% RSLogix 500 project SARANARA_BAK012.RSS, saved by version 8.10.00.18 %
PROJECT "SARANARA"    % processor: MicroLogix 1200 %

PROGRAM FILES
  LAD 2   7 rungs

DATA FILES
  O0 OUTPUT  4 elements
  I1 INPUT  4 elements
  S2 STATUS  66 elements
  B3 BINARY  1 elements
  T4 TIMER  1 elements
  C5 COUNTER  2 elements
  R6 CONTROL  1 elements
  N7 INTEGER  1 elements

LADDER 2
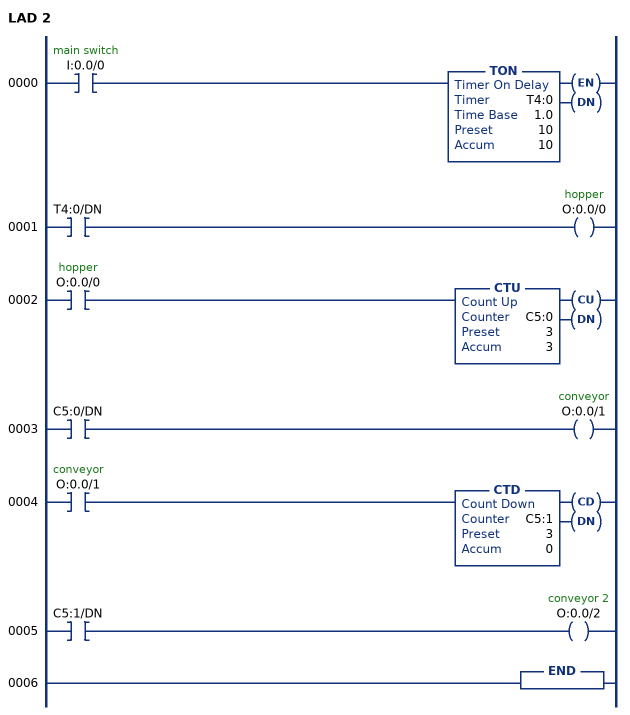
% Rung: 0 %
SOR XIC I:0.0/0 TON T4:0 1.0 10 10 EOR
%   I:0.0/0  "main switch" %
% Rung: 1 %
SOR XIC T4:0/DN OTE O:0.0/0 EOR
%   O:0.0/0  "hopper" %
% Rung: 2 %
SOR XIC O:0.0/0 CTU C5:0 3 3 EOR
%   O:0.0/0  "hopper" %
% Rung: 3 %
SOR XIC C5:0/DN OTE O:0.0/1 EOR
%   O:0.0/1  "conveyor" %
% Rung: 4 %
SOR XIC O:0.0/1 CTD C5:1 3 0 EOR
%   O:0.0/1  "conveyor" %
% Rung: 5 %
SOR XIC C5:1/DN OTE O:0.0/2 EOR
%   O:0.0/2  "conveyor 2" %
% Rung: 6 %
SOR END EOR

DATA TABLE (non-zero values as saved)
DATA T4
% .PRE .ACC %
% T4:0 % 10 10
DATA C5
% .PRE .ACC %
% C5:0 % 3 3
% C5:1 % 3 0
